// Mitsubishi GX Works2 project: PLC 데이터 명령 (대소비교)   PLC: Q03UDV

PROGRAM MAIN
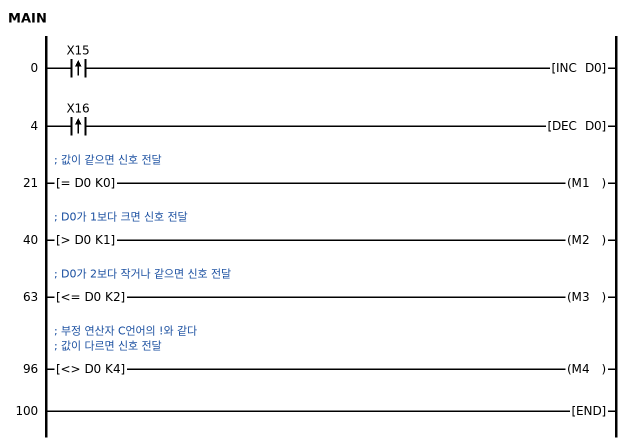
0     LDP     X15
      INC     D0
4     LDP     X16
      DEC     D0
; 값이 같으면 신호 전달
21    LD=     D0 K0
      OUT     M1
; D0가 1보다 크면 신호 전달
40    LD>     D0 K1
      OUT     M2
; D0가 2보다 작거나 같으면 신호 전달
63    LD<=    D0 K2
      OUT     M3
; 부정 연산자 C언어의 !와 같다
; 값이 다르면 신호 전달
96    LD<>    D0 K4
      OUT     M4
100   END
END_PROGRAM
